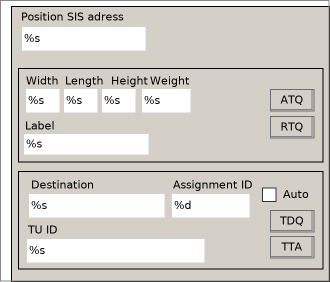
VISUALIZATION V_SIS_Control  // 330x282
VAR_IN_OUT	
	{attribute 'VAR_IN_OUT_AS_POINTER'}
	fb_VizuSIS	: FB_VizuSIS;	
		
END_VAR
    Rectangle (11,6 319x276)
    Textfield (21,26 125x25), "%s", text variable: fb_VizuSIS.PositionString, colour toggle: fb_VizuSIS.BadPosition
        OnMouseClick: write the text variable via Edit
    Label (18,7 117x20), "Position SIS adress"
    Rectangle (18,68 305x94)
    Button (270,89 44x22), "ATQ"
        tap fb_VizuSIS.ATQ
    Textfield (25,88 35x25), "%s", text variable: fb_VizuSIS.ATQ_Dimension.Width
        OnMouseClick: write the text variable via Edit
    Textfield (101,88 35x25), "%s", text variable: fb_VizuSIS.ATQ_Dimension.Height
        OnMouseClick: write the text variable via Edit
    Textfield (63,88 35x25), "%s", text variable: fb_VizuSIS.ATQ_Dimension.Length
        OnMouseClick: write the text variable via Edit
    Textfield (141,88 50x25), "%s", text variable: fb_VizuSIS.ATQ_Dimension.Weight
        OnMouseClick: write the text variable via Edit
    Label (23,71 41x20), "Width"
    Label (62,71 48x20), "Length"
    Label (108,71 41x20), "Height"
    Label (147,71 48x20), "Weight"
    Textfield (23,133 126x22), "%s", text variable: fb_VizuSIS.ATQ_Label
        OnMouseClick: write the text variable via Edit
    Button (270,116 44x22), "RTQ"
        tap fb_VizuSIS.RTQ
    Rectangle (18,171 305x98)
    Button (270,236 44x22), "TTA"
        tap fb_VizuSIS.TTA
    Textfield (28,193 137x25), "%s", text variable: fb_VizuSIS.TTA_Destination
        OnMouseClick: write the text variable via Edit
    Button (270,210 44x22), "TDQ"
        tap fb_VizuSIS.TDQ
    Label (25,220 117x20), "TU ID"
    Textfield (26,238 179x25), "%s", text variable: fb_VizuSIS.TU_ID, input disabled if: fb_VizuSIS.AutoID
        OnMouseClick: write the text variable via Edit, min 18, max 18
    Label (28,175 117x20), "Destination"
    Label (22,116 117x20), "Label"
    Textfield (171,193 79x25), "%d", text variable: fb_VizuSIS.AssignmentID, input disabled if: fb_VizuSIS.AutoID
        OnMouseClick: write the text variable via Edit
    Label (170,175 90x20), "Assignment ID"
    Checkbox (260,183 51x23), "Auto", tooltip "Reuse TU ID and Assignment ID from TU Table", variable: fb_VizuSIS.AutoID
END_VISUALIZATION

(* stored: Version 1.1.0.1, ProductVersion 3.1.4024.9
   Visu V_SIS_Control: Id {6c6a2781-72fb-4d89-846d-4dbdaa225ada} *)
